Staubli VAL3: compose.pgx

public program compose(num x_nIndexTool)
  local trsf tPar
  local tool tGun
  local point pPoint
begin
  pPoint=here(flange,world)
  tPar=!pPoint.trsf*saveData:rif2.trsf
  tGun.trsf=tPar
  call setTool(tGun,x_nIndexTool)
end
